FUNCTION_BLOCK STOPGO (* ECC with no Transient ECC State *)
  (* Standard: 61499-2 *)
  (* Version 0.0, 2018-12-17, JHC, Holobloc Inc *)
  (* Compiler header: package fb.rt.test; *)
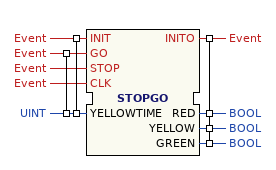
  EVENT_INPUT
    INIT WITH YELLOWTIME; (* Initialization Request *)
    GO WITH YELLOWTIME; (* Normal Execution Request *)
    STOP;
    CLK;
  END_EVENT
  EVENT_OUTPUT
    INITO WITH RED, YELLOW, GREEN; (* Initialization Confirm *)
  END_EVENT
  VAR_INPUT
    YELLOWTIME : UINT; (* Input event qualifier *)
  END_VAR
  VAR_OUTPUT
    RED : BOOL; (* Output event qualifier *)
    YELLOW : BOOL;
    GREEN : BOOL;
  END_VAR
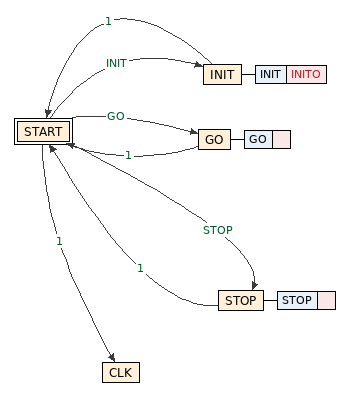
  EC_STATES
    START; (* Initial State *)
    INIT : INIT -> INITO; (* Initialization *)
    GO : GO;
    STOP : STOP;
    CLK;
  END_STATES
  EC_TRANSITIONS
    INIT TO START := 1;
    START TO INIT := INIT;
    START TO GO := GO;
    GO TO START := 1;
    START TO STOP := STOP;
    STOP TO START := 1;
    START TO CLK := 1;
  END_TRANSITIONS
  ALGORITHM INIT IN ST: (* Initialization algorithm *)
RED:=FALSE;
YELLOW:=FALSE;
GREEN:=FALSE;
  END_ALGORITHM
  ALGORITHM STOP IN ST:

  END_ALGORITHM
  ALGORITHM GO IN ST:

  END_ALGORITHM
  ALGORITHM CLK IN ST:

  END_ALGORITHM
END_FUNCTION_BLOCK
